(* CoDeSys 2.3.9.41 project: Mixer1_CFC_IL_LD_SFC_ST_v8.pro *)
(* Libraries: Standard.lib 4.10.05 12:14:46, IecSfc.lib 13.4.06 16:51:28, SYSLIBCALLBACK.LIB 26.9.08 17:43:52 *)

(* Task configuration *)
TASK NewTask (PRIORITY := 1); (* freewheeling *)
	VIS_PRG();
	PLC_Timers();
	PLC_ST_PRG();
END_TASK

(* Global variable list: Global_Variables *)
VAR_GLOBAL  (* 13 входов на 14 выходов + всп. пер. + входы и выходы таймеров  *)
(* Входы *)
    (* Кнопки Push Buttons -- префикс pb *)
	pbStrt: BOOL;             (* кнопка "Пуск"                                  *)
    pbStop: BOOL;             (* кнопка "Стоп"                                  *)
	pbCmpl: BOOL;             (* кнопка "Завершение работы"                     *)
	(* Кнопки-переключатели Switch Buttons -- префикс sb *)
	sbEVlv: BOOL;             (* переключатель "Открыть аварийный клапан"       *)
    (* Датчики Sensors -- префикс s *)
	sT1, _sT1: BOOL;          (* датчик нулевого уровня бака 1                  *)
	sT2, _sT2: BOOL;          (* датчик нулевого уровня бака 2                  *)
	sL0      : BOOL;          (* датчик уровня 0 резервуара                     *)
	sL1      : BOOL;          (* датчик уровня 1 резервуара                     *)
	sL2      : BOOL;          (* датчик уровня 2 резервуара                     *)
	sM,  _sM : BOOL;          (* датчик работы привода мешалки                  *)
	sUT      : BOOL;          (* датчик верхней температуры нагревателя         *)
	sLT      : BOOL;          (* датчик нижней  температуры нагревателя         *)
	sWT, _sWT: BOOL;          (* датчик рабочей температуры нагревателя         *)
(* Выходы *)
	(* Клапаны/Лампы Valves/Lamps -- префикс vlv/lmp *)
	vlv1, _vlv1: BOOL;        (* открыть клапан 1                               *)
	vlv2, _vlv2: BOOL;        (* открыть клапан 2                               *)
	vlvP       : BOOL;        (* открыть разливной клапан                       *)
	vlvE, _vlvE: BOOL;        (* открыть аварийный клапан                       *)
	(* Приводы/Лампы Actuators/Lamps -- префикс act/lmp *)
 	actHtr, _actHtr: BOOL;    (* включить нагреватель                           *)
	actMtr, _actMtr: BOOL;    (* запустить привод мешалки                       *)
    (* Режимы/Состояния/Лампы Modes/States/Lamps -- префикс m/q/lmp *)
	mSysOn,  _mSysOn : BOOL;  (* система включена                               *)
	mCompl,  _mCompl : BOOL;  (* режим плавного завершения работы установки     *)
    mMxIsFn, _mMxIsFn: BOOL;  (* смесь приготовлена                             *)
    mMxIsBd, _mMxIsBd: BOOL;  (* смесь испорчена                                *)
    mC1InMx, _mC1InMx: BOOL;  (* в смеси есть компонент 1                       *)
    mC2InMx, _mC2InMx: BOOL;  (* в смеси есть компонент 2                       *)
    (* Ошибки/Лампы Errors/Lamps -- префикс err/lmp *)
	errHtr, _errHtr: BOOL;    (* сигнал ошибки нагревателя                      *)
	errMtr, _errMtr: BOOL;    (* сигнал ошибки привода мешалки                  *)
(* Вспомогательные переменные Conditions -- префикс c *)
	cFin: BOOL;               (* условие завершения работы установки            *)
(* Таймеры Timers -- префикс tmr *)
	tmrMtr: TON := (PT := T#2s);    (* таймер ожидания запуска мешалки          *)
    tmrMix: TON := (PT := T#7s);    (* таймер работы мешалки                    *)
    tmrHtr: TON := (PT := T#12s);   (* таймер ожидания нагрева                  *)
END_VAR

(* POU VIS_PRG, ST *)
PROGRAM VIS_PRG
VAR
  (* ------- Обычные кнопки ------- *)
  PBTnk1: BOOL;                  (* наполнить бак 1 (синий)                *)
  PBTnk2: BOOL;                  (* наполнить бак 2 (красный)              *)
  PBCmp1: BOOL;                  (* осушить бак 1                          *)
  PBCmp2: BOOL;                  (* осушить бак 2                          *)
  (* ------- Кнопки-переключатели ------- *)
  SBMtrBrk: BOOL;                (* поломка привода мешалки                *)
  SBHtrBrk: BOOL;                (* поломка нагревателя                    *)
  (* ------- Жидкости ------- *)
  Cmp1, _Cmp1: INT;              (* объем компонента 1 (синего)   в баке 1 *)
  Cmp2, _Cmp2: INT;              (* объем компонента 2 (красного) в баке 2 *)
  Mix,   _Mix: INT;              (* объем смеси в резервуаре               *)
  MixClr:      DWORD;            (* цвет  смеси в резервуаре               *)
  Red,   _Red: REAL;             (* коэффициент красного цвета в смеси     *)
  (* ------- Нагреватель ------- *)
  HtrClr: DWORD:=16#00_FF_FF_FF; (* температура нагревателя (цвет)         *)
  HtrRed, _HtrRed: BYTE;         (* степень накаливания нагревателя        *)
  HtrOn: BOOL;                   (* нагреватель функционирует (греет)      *)
END_VAR
(* объем каждого из баков --- 300 единиц *)
(* пропускная способность каждого клапана равняется 1 единице за время прохода рабочего цикла ПЛК *)
(* но отрисовывать уменьшение объема жидкости в баке нужно в 3 раза медленне, чем происходит отрисовка заполнеия резервуара для смешивания *)
(* считается, что все клапаны обладают одинаковой пропускной способностью *)
Cmp1:= MAX(0,MIN(360,BOOL_TO_INT(NOT PBCmp1)*_Cmp1+BOOL_TO_INT(PBTnk1)*360-BOOL_TO_INT(vlv1)));
Cmp2:= MAX(0,MIN(240,BOOL_TO_INT(NOT PBCmp2)*_Cmp2+BOOL_TO_INT(PBTnk2)*240-BOOL_TO_INT(vlv2)));
Mix := MAX(0,_Mix
             +BOOL_TO_INT(vlv1 AND _Cmp1>0)
             +BOOL_TO_INT(vlv2 AND _Cmp2>0)
             -BOOL_TO_INT(vlvE AND _Mix >0)
             -BOOL_TO_INT(vlvP AND _Mix >0)
          );
Red := BOOL_TO_INT(Mix>0)*(_Red*_Mix+1*BOOL_TO_INT(vlv2 AND _Cmp2>0)
                                    -1*_Red*BOOL_TO_INT(vlvP AND _Mix >0)
                                    -1*_Red*BOOL_TO_INT(vlvE AND _Mix >0)
                                                                         )/MAX(1,Mix);
MixClr := 65536*REAL_TO_BYTE(255*(1-Red))+REAL_TO_BYTE(255*Red);
(* ------- Нагреватель ------- *)
HtrOn:=actHtr AND NOT SBHtrBrk; (* нагреватель включается, если не сломан       *)
HtrRed:=_HtrRed+BOOL_TO_BYTE(HtrOn AND _HtrRed<255)-BOOL_TO_BYTE(NOT HtrOn AND _HtrRed>0);
HtrClr:=65536*(255-HtrRed)+256*(255-HtrRed)+255;
(* ------- Выставление сигналов датчиков ------- *)
sT1:=(Cmp1>0);                  (* датчик нулевого уровня бака 1                *)
sT2:=(Cmp2>0);                  (* датчик нулевого уровня бака 2                *)
sL0:=(Mix>0);                   (* датчик уровня 0 резервуара                   *)
sL1:=(Mix>=180);                (* датчик уровня 1 резервуара                   *)
sL2:=(Mix>=300);                (* датчик уровня 2 резервуара                   *)
sM := NOT SBMtrBrk AND actMtr;  (* привод мешалки включается, если не сломан    *)
sUT:=(HtrRed>=252);
sLT:=(HtrRed>=160);
sWT:=(HtrRed>=150);
(* -------  Псевдооператорный раздел ------- *)
_Cmp1:=Cmp1; _Cmp2:=Cmp2; _Mix:=Mix; _Red:=Red; _HtrRed:=HtrRed;
END_PROGRAM

(* POU PLC_Timers, FBD *)
PROGRAM PLC_Timers
VAR
END_VAR
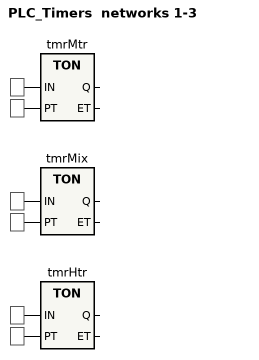
_FBD_ (* Function Block Diagram *)
NETWORK 1
	tmrMtr:TON(IN: , PT: )
NETWORK 2
	tmrMix:TON(IN: , PT: )
NETWORK 3
	tmrHtr:TON(IN: , PT: )
_END_FBD_
END_PROGRAM

(* POU PLC_ST_PRG, ST *)
PROGRAM PLC_ST_PRG
VAR
END_VAR
(* ------- Ошибки/Лампы ------- *)
IF NOT _errHtr AND NOT sWT AND (tmrHtr.Q OR _actHtr AND _sWT) THEN errHtr:=1;         (* errHtr+  *)
ELSIF  _errHtr AND pbStop                                     THEN errHtr:=0;         (* errHtr-  *)
END_IF;
IF NOT _errMtr AND NOT sM AND (tmrMtr.Q OR _actMtr AND _sM) THEN errMtr:=1;           (* errMtr+  *)
ELSIF  _errMtr AND pbStop                                   THEN errMtr:=0;           (* errMtr-  *)
END_IF;
(* ------- Режимы/Состояния/Лампы ------- *)
IF NOT _mMxIsBd AND     sL0 AND _vlvE AND _mC2InMx AND NOT _mMxIsFn THEN mMxIsBd:=1;  (* mMxIsBd+ *)
ELSIF  _mMxIsBd AND NOT sL0                                         THEN mMxIsBd:=0;  (* mMxIsBd- *)
END_IF;
IF NOT _mMxIsFn AND     sL0 AND NOT mMxIsBd AND tmrMix.Q THEN mMxIsFn:=1;             (* mMxIsFn+ *)
ELSIF  _mMxIsFn AND NOT sL0                              THEN mMxIsFn:=0;             (* mMxIsFn- *)
END_IF;
IF NOT _mC1InMx AND     sL0 AND _vlv1 AND _sT1 THEN mC1InMx:=1;                       (* mC1InMx+ *)
ELSIF  _mC1InMx AND NOT sL0                    THEN mC1InMx:=0;                       (* mC1InMx- *)
END_IF;
IF NOT _mC2InMx AND     sL0 AND _vlv2 AND _sT2 THEN mC2InMx:=1;                       (* mC2InMx+ *)
ELSIF  _mC2InMx AND NOT sL0                    THEN mC2InMx:=0;                       (* mC2InMx- *)
END_IF;
(* ------- Вспомогательные переменные ------- *)
cFin:= _mCompl AND NOT _vlv1 AND NOT sL0
                OR errHtr OR errMtr OR mMxIsBd OR sbEVlv OR pbStop
                OR NOT sT1 AND NOT sL1 AND NOT mMxIsFn
                OR NOT sT2 AND NOT sL2 AND NOT mMxIsFn;                               (* cFin     *)
(* ------- Режимы/Состояния/Лампы ------- *)
IF NOT _mSysOn AND pbStrt AND NOT cFin THEN mSysOn:=1;                                (* mSysOn+  *)
ELSIF  _mSysOn AND                cFin THEN mSysOn:=0;                                (* mSysOn-  *)
END_IF;
IF NOT _mCompl AND     mSysOn AND pbCmpl THEN mCompl:=1;                              (* mCompl+  *)
ELSIF  _mCompl AND NOT mSysOn            THEN mCompl:=0;                              (* mCompl-  *)
END_IF;
(* ------- Нагреватель/Лампа ------- *)
IF NOT _actHtr AND      mSysOn AND NOT sLT  THEN actHtr:=1;                           (* actHtr+  *)
ELSIF  _actHtr AND (NOT mSysOn OR      sUT) THEN actHtr:=0;                           (* actHtr-  *)
END_IF;
(* ------- Клапаны/Приводы/Лампы ------- *)
vlv1:=mSysOn AND sT1 AND NOT sL1               AND NOT mC2InMx AND sWT;               (* vlv1     *)
Vlv2:=mSysOn AND sT2 AND     sL1   AND NOT sL2 AND NOT mMxIsFn AND sWT;               (* vlv2     *)
actMtr:=mSysOn AND mC1InMx AND mC2InMx AND sL2 AND NOT mMxIsFn AND sWT;               (* actMtr   *)
vlvP:=mSysOn AND mMxIsFn;                                                             (* vlvP     *)
vlvE:=sbEVlv;                                                                         (* vlvE     *)
(* ------- Раздел таймеров ------- *)
tmrHtr.IN:= actHtr AND NOT sWT;                                                      (* tmrHtr.IN *)
tmrMtr.IN:= actMtr AND NOT sM;                                                       (* tmrMtr.IN *)
tmrMix.IN:= actMtr AND     sM;                                                       (* tmrMix.IN *)
(* ------- Псевдооператорный раздел ------- *)
_errMtr:=errMtr; _errHtr:=errHtr;
_mC1InMx:=mC1InMx; _mC2InMx:=mC2InMx;
_mMxIsFn:=mMxIsFn; _mMxIsBd:=mMxIsBd;
_mSysOn:=mSysOn; _mCompl:=mCompl;
_vlvE:=vlvE; _vlv1:=vlv1; _vlv2:=vlv2;
_actHtr:=actHtr; _actMtr:=actMtr;
_sT1:=sT1; _sT2:=sT2; _sM :=sM; _sWT:=sWT;
END_PROGRAM

(* POU PLC_CFC_PRG, FAI *)
PROGRAM PLC_CFC_PRG
VAR
END_VAR
(* body not read: cfc101 *)
END_PROGRAM

(* POU PLC_IL_PRG, IL *)
PROGRAM PLC_IL_PRG
VAR
END_VAR
	(* ------- Ошибки/Лампы ------- *)
	(* IF      *)
	LDN		_errHtr							(* errHtr  *)
	ANDN	sWT
	AND		(tmrHtr.Q
	OR		(_actHtr
	AND		_sWT
	)
	)
	S		errHtr		(* errHtr:=1 *)
	LD		_errHtr		(* ELSIF     *)
	AND		pbStop
	R		errHtr		(* errHtr:=0 *)
	(* END_IF  *)
	(* ------- *)
	(* IF      *)
	LDN		_errMtr							(* errMtr  *)
	ANDN	sM
	AND		(tmrMtr.Q
	OR		(_actMtr
	AND		_sM
	)
	)
	S		errMtr		(* errMtr:=1 *)
	LD		_errMtr		(* ELSIF     *)
	AND		pbStop
	R		errMtr		(* errMtr:=0 *)
	(* END_IF  *)
	(* ------- Режимы/Состояния/Лампы ------- *)
	(* IF      *)
	LDN		_mMxIsBd						(* mMxIsBd *)
	AND		sL0
	AND		_vlvE
	AND		_mC2InMx
	ANDN	_mMxIsFn
	S		mMxIsBd		(* mMxIsBd:=1 *)
	LD		_mMxIsBd	(* ELSIF      *)
	ANDN	sL0
	R		mMxIsBd 	(* mMxIsBd:=0 *)
	(* END_IF  *)
	(* ------- *)
	(* IF      *)
	LDN		_mMxIsFn						(* mMxIsFn *)
	AND		sL0
	ANDN	mMxIsBd
	AND		tmrMix.Q
	S		mMxIsFn		(* mMxIsFn:=1 *)
	LD		_mMxIsFn	(* ELSIF      *)
	ANDN	sL0
	R		mMxIsFn		(* mMxIsFn:=0 *)
	(* END_IF  *)
	(* ------- *)
	(* IF      *)
	LDN		_mC1InMx						(* mC1InMx *)
	AND		sL0
	AND		_vlv1
	AND		_sT1
	S		mC1InMx		(* mC1InMx:=1 *)
	LD		_mC1InMx	(* ELSIF      *)
	ANDN	sL0
	R		mC1InMx		(* mC1InMx:=0 *)
	(* END_IF  *)
	(* ------- *)
	(* IF      *)
	LDN		_mC2InMx						(* mC2InMx *)
	AND		sL0
	AND		_vlv2
	AND		_sT2
	S		mC2InMx		(* mC2InMx:=1 *)
	LD		_mC2InMx	(* ELSIF      *)
	ANDN	sL0
	R		mC2InMx		(* mC2InMx:=0 *)
	(* END_IF  *)
	(* ------- Вспомогательные переменные ------- *)
	LD		_mCompl							(* cFin    *)
	ANDN	_vlv1
	ANDN	sL0
	OR		errHtr
	OR		errMtr
	OR		mMxIsBd
	OR		sbEVlv
	OR		pbStop
	OR		(sT1
	NOT
	ANDN	sL1
	ANDN	mMxIsFn
	)
	OR		(sT2
	NOT
	ANDN	sL2
	ANDN	mMxIsFn
	)
	ST		cFin
	(* ------- Режимы/Состояния/Лампы ------- *)
	(* IF      *)
	LDN		_mSysOn							(* mSysOn  *)
	AND		pbStrt
	ANDN	cFin
	S		mSysOn		(* mSysOn:=1 *)
	LD		_mSysOn		(* ELSIF     *)
	AND		cFin
	R		mSysOn		(* mSysOn:=0 *)
	(* END_IF  *)
	(* ------- *)
	(* IF      *)
	LDN		_mCompl							(* mCompl  *)
	AND		mSysOn
	AND		pbCmpl
	S		mCompl		(* mCompl:=1 *)
	LD		_mCompl		(* ELSIF     *)
	ANDN	mSysOn
	R		mCompl		(* mCompl:=0 *)
	(* END_IF  *)
	(* ------- Нагреватель/Лампа ------- *)
	(* IF      *)
	LDN		_actHtr							(* actHtr  *)
	AND		mSysOn
	ANDN	sLT
	S		actHtr		(* actHtr:=1 *)
	LD		_actHtr		(* ELSIF     *)
	AND		(mSysOn
	NOT
	OR		sUT
	)
	R		actHtr		(* actHtr:=0 *)
	(* END_IF  *)
	(* ------- Клапаны/Лампы ------- *)
	LD		mSysOn 						    (* Vlv1    *)
	AND		sT1
	ANDN	sL1
	ANDN	mC2InMx
	AND		sWT
	ST		vlv1
	(* ------- Клапаны/Лампы ------- *)
	LD		mSysOn 							(* Vlv2    *)
	AND		sT2
	AND		sL1
	ANDN	sL2
	ANDN	mMxIsFn
	AND		sWT
	ST		vlv2
	(* ------- Приводы/Лампы ------- *)
	LD		mSysOn							(* actMtr  *)
	AND		mC1InMx
	AND		mC2InMx
	AND		sL2
	ANDN	mMxIsFn
	AND		sWT
	ST		actMtr
	(* ------- Клапаны/Лампы ------- *)
	LD		mSysOn							(* vlvP    *)
	AND		mMxIsFn
	ST		vlvP
	(* ------- *)
	LD		sbEVlv							(* vlvE    *)
	ST		vlvE
	(* ------- Раздел таймеров ------- *)
	LD		actHtr						  (* tmrHtr.IN *)
	ANDN	sWT
	ST		tmrHtr.IN
	(* ------- *)
	LD		actMtr						  (* tmrMtr.IN *)
	ANDN	sM
	ST		tmrMtr.IN
	(* ------- *)
	LD		actMtr						  (* tmrMix.IN *)
	AND		sM
	ST		tmrMix.IN
	(* ------- Псевдооператорный раздел ------- *)
	(* ------- Ошибки ------- *)
	LD		errMtr
	ST		_errMtr		(* _errMtr:=errMtr;   *)
	LD		errHtr
	ST		_errHtr		(* _errHtr:=errHtr;   *)
	(* ------- Режимы/Состояния ------- *)
	LD		mC1InMx
	ST		_mC1InMx	(* _mC1InMx:=mC1InMx; *)
	LD		mC2InMx
	ST		_mC2InMx	(* _mC2InMx:=mC2InMx; *)
	LD		mMxIsFn
	ST		_mMxIsFn	(* _mMxIsFn:=mMxIsFn; *)
	LD		mMxIsBd
	ST		_mMxIsBd	(* _mMxIsBd:=mMxIsBd; *)
	LD		mSysOn
	ST		_mSysOn		(* _mSysOn:=mSysOn;   *)
	LD		mCompl
	ST		_mCompl		(* _mCompl:=mCompl;   *)
	(* ------- Клапаны ------- *)
	LD		vlvE
	ST		_vlvE		(* _vlvE:=vlvE;       *)
	LD		vlv1
	ST		_vlv1		(* _vlv1:=vlv1;       *)
	LD		vlv2
	ST		_vlv2		(* _vlv2:=vlv2;       *)
	(* ------- Приводы ------- *)
	LD		actHtr
	ST		_actHtr		(* _actHtr:=actHtr;   *)
	LD		actMtr
	ST		_actMtr		(* _actMtr:=actMtr;   *)
	(* ------- Датчики ------- *)
	LD		sT1
	ST		_sT1		(* _sT1:=sT1;         *)
	LD		sT2
	ST		_sT2		(* _sT2:=sT2;         *)
	LD		sM
	ST		_sM			(* _sM:=sM;           *)
	LD		sWT
	ST		_sWT		(* _sWT:=sWT;         *)
END_PROGRAM

(* POU PLC_LD_PRG, LD *)
PROGRAM PLC_LD_PRG
VAR
END_VAR
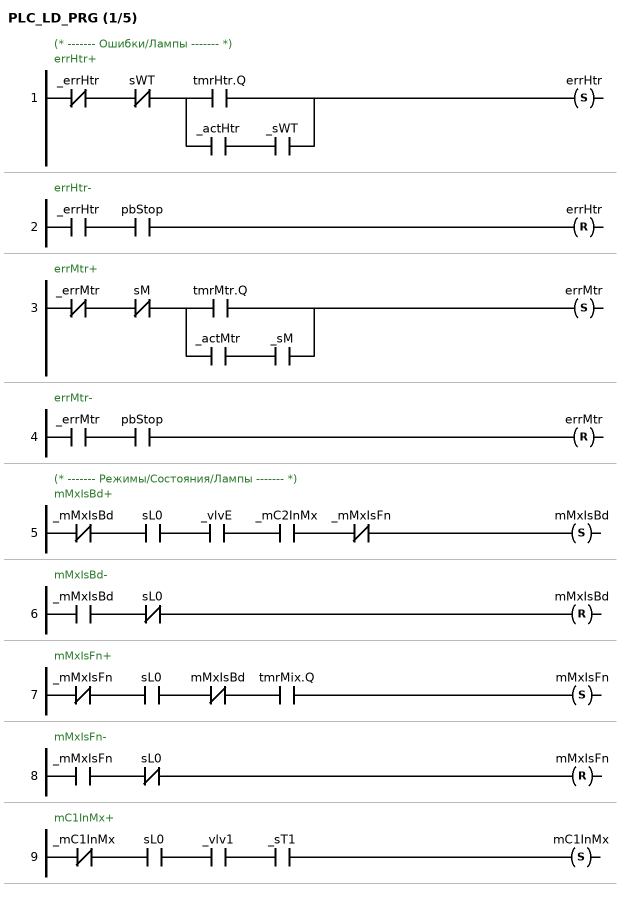
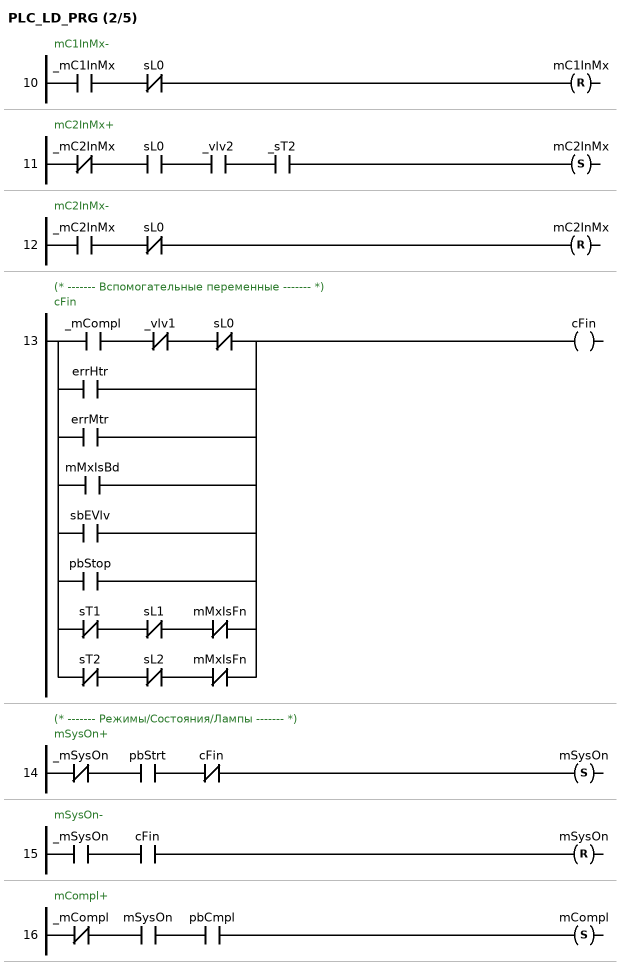
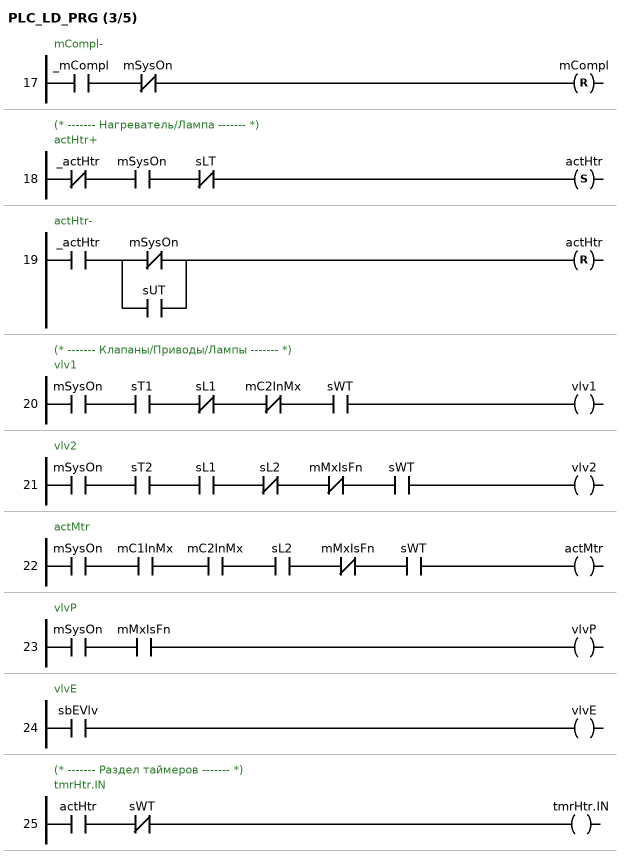
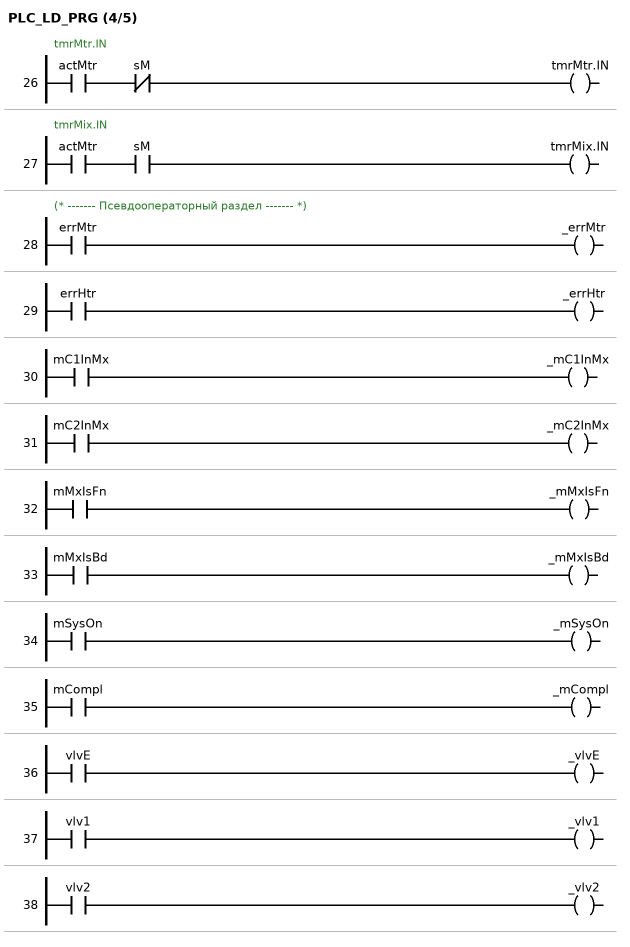
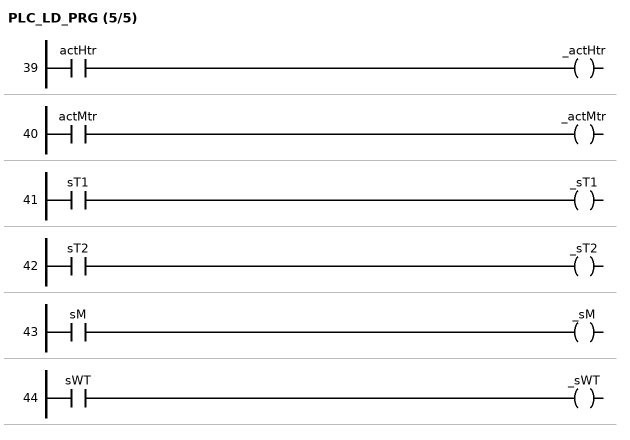
_LD_ (* Ladder Diagram *)
NETWORK 1 (* ( * ------- Ошибки/Лампы ------- * ) / errHtr+ *)
	[/_errHtr] - [/sWT] - { [tmrHtr.Q] | [_actHtr] - [_sWT] } --- (S errHtr)
NETWORK 2 (* errHtr- *)
	[_errHtr] - [pbStop] --- (R errHtr)
NETWORK 3 (* errMtr+ *)
	[/_errMtr] - [/sM] - { [tmrMtr.Q] | [_actMtr] - [_sM] } --- (S errMtr)
NETWORK 4 (* errMtr- *)
	[_errMtr] - [pbStop] --- (R errMtr)
NETWORK 5 (* ( * ------- Режимы/Состояния/Лампы ------- * ) / mMxIsBd+ *)
	[/_mMxIsBd] - [sL0] - [_vlvE] - [_mC2InMx] - [/_mMxIsFn] --- (S mMxIsBd)
NETWORK 6 (* mMxIsBd- *)
	[_mMxIsBd] - [/sL0] --- (R mMxIsBd)
NETWORK 7 (* mMxIsFn+ *)
	[/_mMxIsFn] - [sL0] - [/mMxIsBd] - [tmrMix.Q] --- (S mMxIsFn)
NETWORK 8 (* mMxIsFn- *)
	[_mMxIsFn] - [/sL0] --- (R mMxIsFn)
NETWORK 9 (* mC1InMx+ *)
	[/_mC1InMx] - [sL0] - [_vlv1] - [_sT1] --- (S mC1InMx)
NETWORK 10 (* mC1InMx- *)
	[_mC1InMx] - [/sL0] --- (R mC1InMx)
NETWORK 11 (* mC2InMx+ *)
	[/_mC2InMx] - [sL0] - [_vlv2] - [_sT2] --- (S mC2InMx)
NETWORK 12 (* mC2InMx- *)
	[_mC2InMx] - [/sL0] --- (R mC2InMx)
NETWORK 13 (* ( * ------- Вспомогательные переменные ------- * ) / cFin *)
	{ [_mCompl] - [/_vlv1] - [/sL0] | [errHtr] | [errMtr] | [mMxIsBd] | [sbEVlv] | [pbStop] | [/sT1] - [/sL1] - [/mMxIsFn] | [/sT2] - [/sL2] - [/mMxIsFn] } --- (cFin)
NETWORK 14 (* ( * ------- Режимы/Состояния/Лампы ------- * ) / mSysOn+ *)
	[/_mSysOn] - [pbStrt] - [/cFin] --- (S mSysOn)
NETWORK 15 (* mSysOn- *)
	[_mSysOn] - [cFin] --- (R mSysOn)
NETWORK 16 (* mCompl+ *)
	[/_mCompl] - [mSysOn] - [pbCmpl] --- (S mCompl)
NETWORK 17 (* mCompl- *)
	[_mCompl] - [/mSysOn] --- (R mCompl)
NETWORK 18 (* ( * ------- Нагреватель/Лампа ------- * ) / actHtr+ *)
	[/_actHtr] - [mSysOn] - [/sLT] --- (S actHtr)
NETWORK 19 (* actHtr- *)
	[_actHtr] - { [/mSysOn] | [sUT] } --- (R actHtr)
NETWORK 20 (* ( * ------- Клапаны/Приводы/Лампы ------- * ) / vlv1 *)
	[mSysOn] - [sT1] - [/sL1] - [/mC2InMx] - [sWT] --- (vlv1)
NETWORK 21 (* vlv2 *)
	[mSysOn] - [sT2] - [sL1] - [/sL2] - [/mMxIsFn] - [sWT] --- (vlv2)
NETWORK 22 (* actMtr *)
	[mSysOn] - [mC1InMx] - [mC2InMx] - [sL2] - [/mMxIsFn] - [sWT] --- (actMtr)
NETWORK 23 (* vlvP *)
	[mSysOn] - [mMxIsFn] --- (vlvP)
NETWORK 24 (* vlvE *)
	[sbEVlv] --- (vlvE)
NETWORK 25 (* ( * ------- Раздел таймеров ------- * ) / tmrHtr.IN *)
	[actHtr] - [/sWT] --- (tmrHtr.IN)
NETWORK 26 (* tmrMtr.IN *)
	[actMtr] - [/sM] --- (tmrMtr.IN)
NETWORK 27 (* tmrMix.IN *)
	[actMtr] - [sM] --- (tmrMix.IN)
NETWORK 28 (* ( * ------- Псевдооператорный раздел ------- * ) *)
	[errMtr] --- (_errMtr)
NETWORK 29
	[errHtr] --- (_errHtr)
NETWORK 30
	[mC1InMx] --- (_mC1InMx)
NETWORK 31
	[mC2InMx] --- (_mC2InMx)
NETWORK 32
	[mMxIsFn] --- (_mMxIsFn)
NETWORK 33
	[mMxIsBd] --- (_mMxIsBd)
NETWORK 34
	[mSysOn] --- (_mSysOn)
NETWORK 35
	[mCompl] --- (_mCompl)
NETWORK 36
	[vlvE] --- (_vlvE)
NETWORK 37
	[vlv1] --- (_vlv1)
NETWORK 38
	[vlv2] --- (_vlv2)
NETWORK 39
	[actHtr] --- (_actHtr)
NETWORK 40
	[actMtr] --- (_actMtr)
NETWORK 41
	[sT1] --- (_sT1)
NETWORK 42
	[sT2] --- (_sT2)
NETWORK 43
	[sM] --- (_sM)
NETWORK 44
	[sWT] --- (_sWT)
_END_LD_
(* the same logic as Structured Text *)
(* Network 1: ( * ------- Ошибки/Лампы ------- * ) / errHtr+ *)
IF NOT _errHtr AND NOT sWT AND (tmrHtr.Q OR _actHtr AND _sWT) THEN errHtr := TRUE; END_IF;
(* Network 2: errHtr- *)
IF _errHtr AND pbStop THEN errHtr := FALSE; END_IF;
(* Network 3: errMtr+ *)
IF NOT _errMtr AND NOT sM AND (tmrMtr.Q OR _actMtr AND _sM) THEN errMtr := TRUE; END_IF;
(* Network 4: errMtr- *)
IF _errMtr AND pbStop THEN errMtr := FALSE; END_IF;
(* Network 5: ( * ------- Режимы/Состояния/Лампы ------- * ) / mMxIsBd+ *)
IF NOT _mMxIsBd AND sL0 AND _vlvE AND _mC2InMx AND NOT _mMxIsFn THEN mMxIsBd := TRUE; END_IF;
(* Network 6: mMxIsBd- *)
IF _mMxIsBd AND NOT sL0 THEN mMxIsBd := FALSE; END_IF;
(* Network 7: mMxIsFn+ *)
IF NOT _mMxIsFn AND sL0 AND NOT mMxIsBd AND tmrMix.Q THEN mMxIsFn := TRUE; END_IF;
(* Network 8: mMxIsFn- *)
IF _mMxIsFn AND NOT sL0 THEN mMxIsFn := FALSE; END_IF;
(* Network 9: mC1InMx+ *)
IF NOT _mC1InMx AND sL0 AND _vlv1 AND _sT1 THEN mC1InMx := TRUE; END_IF;
(* Network 10: mC1InMx- *)
IF _mC1InMx AND NOT sL0 THEN mC1InMx := FALSE; END_IF;
(* Network 11: mC2InMx+ *)
IF NOT _mC2InMx AND sL0 AND _vlv2 AND _sT2 THEN mC2InMx := TRUE; END_IF;
(* Network 12: mC2InMx- *)
IF _mC2InMx AND NOT sL0 THEN mC2InMx := FALSE; END_IF;
(* Network 13: ( * ------- Вспомогательные переменные ------- * ) / cFin *)
cFin := _mCompl AND NOT _vlv1 AND NOT sL0 OR errHtr OR errMtr OR mMxIsBd OR sbEVlv OR pbStop OR NOT sT1 AND NOT sL1 AND NOT mMxIsFn OR NOT sT2 AND NOT sL2 AND NOT mMxIsFn;
(* Network 14: ( * ------- Режимы/Состояния/Лампы ------- * ) / mSysOn+ *)
IF NOT _mSysOn AND pbStrt AND NOT cFin THEN mSysOn := TRUE; END_IF;
(* Network 15: mSysOn- *)
IF _mSysOn AND cFin THEN mSysOn := FALSE; END_IF;
(* Network 16: mCompl+ *)
IF NOT _mCompl AND mSysOn AND pbCmpl THEN mCompl := TRUE; END_IF;
(* Network 17: mCompl- *)
IF _mCompl AND NOT mSysOn THEN mCompl := FALSE; END_IF;
(* Network 18: ( * ------- Нагреватель/Лампа ------- * ) / actHtr+ *)
IF NOT _actHtr AND mSysOn AND NOT sLT THEN actHtr := TRUE; END_IF;
(* Network 19: actHtr- *)
IF _actHtr AND (NOT mSysOn OR sUT) THEN actHtr := FALSE; END_IF;
(* Network 20: ( * ------- Клапаны/Приводы/Лампы ------- * ) / vlv1 *)
vlv1 := mSysOn AND sT1 AND NOT sL1 AND NOT mC2InMx AND sWT;
(* Network 21: vlv2 *)
vlv2 := mSysOn AND sT2 AND sL1 AND NOT sL2 AND NOT mMxIsFn AND sWT;
(* Network 22: actMtr *)
actMtr := mSysOn AND mC1InMx AND mC2InMx AND sL2 AND NOT mMxIsFn AND sWT;
(* Network 23: vlvP *)
vlvP := mSysOn AND mMxIsFn;
(* Network 24: vlvE *)
vlvE := sbEVlv;
(* Network 25: ( * ------- Раздел таймеров ------- * ) / tmrHtr.IN *)
tmrHtr.IN := actHtr AND NOT sWT;
(* Network 26: tmrMtr.IN *)
tmrMtr.IN := actMtr AND NOT sM;
(* Network 27: tmrMix.IN *)
tmrMix.IN := actMtr AND sM;
(* Network 28: ( * ------- Псевдооператорный раздел ------- * ) *)
_errMtr := errMtr;
(* Network 29 *)
_errHtr := errHtr;
(* Network 30 *)
_mC1InMx := mC1InMx;
(* Network 31 *)
_mC2InMx := mC2InMx;
(* Network 32 *)
_mMxIsFn := mMxIsFn;
(* Network 33 *)
_mMxIsBd := mMxIsBd;
(* Network 34 *)
_mSysOn := mSysOn;
(* Network 35 *)
_mCompl := mCompl;
(* Network 36 *)
_vlvE := vlvE;
(* Network 37 *)
_vlv1 := vlv1;
(* Network 38 *)
_vlv2 := vlv2;
(* Network 39 *)
_actHtr := actHtr;
(* Network 40 *)
_actMtr := actMtr;
(* Network 41 *)
_sT1 := sT1;
(* Network 42 *)
_sT2 := sT2;
(* Network 43 *)
_sM := sM;
(* Network 44 *)
_sWT := sWT;
END_PROGRAM

(* POU PLC_SFC_PRG, SFC *)
PROGRAM PLC_SFC_PRG
VAR
END_VAR
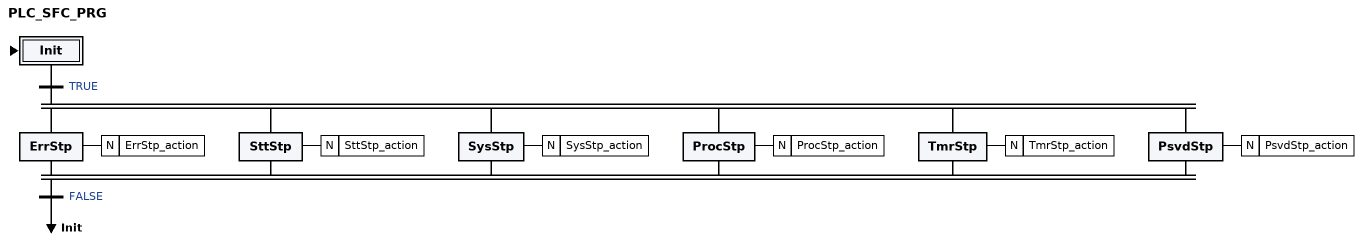
INITIAL_STEP Init:
END_STEP
TRANSITION FROM Init TO (ErrStp, SttStp, SysStp, ProcStp, TmrStp, PsvdStp) := TRUE;
END_TRANSITION
STEP ErrStp:
	ErrStp_action(N);
END_STEP
STEP SttStp:
	SttStp_action(N);
END_STEP
STEP SysStp:
	SysStp_action(N);
END_STEP
STEP ProcStp:
	ProcStp_action(N);
END_STEP
STEP TmrStp:
	TmrStp_action(N);
END_STEP
STEP PsvdStp:
	PsvdStp_action(N);
END_STEP
TRANSITION FROM (ErrStp, SttStp, SysStp, ProcStp, TmrStp, PsvdStp) TO Init := FALSE;
END_TRANSITION

ACTION ErrStp_action:
(* ------- Состояния/Ошибки/Лампы ------- *)
IF NOT _errHtr AND NOT sWT AND (tmrHtr.Q OR _actHtr AND _sWT) THEN errHtr:=1;    (* errHtr+ *)
ELSIF  _errHtr AND pbStop                                     THEN errHtr:=0;    (* errHtr- *)
END_IF;
IF NOT _errMtr AND NOT sM AND (tmrMtr.Q OR _actMtr AND _sM) THEN errMtr:=1;      (* errMtr+ *)
ELSIF  _errMtr AND pbStop                                   THEN errMtr:=0;      (* MtrErr- *)
END_IF;
END_ACTION

ACTION SttStp_action:
(* ------- Состояния/Лампы ------- *)
IF NOT _mMxIsBd AND     sL0 AND _vlvE AND _mC2InMx AND NOT _mMxIsFn THEN mMxIsBd:=1; (* mMxIsBd+ *)
ELSIF  _mMxIsBd AND NOT sL0                                         THEN mMxIsBd:=0; (* mMxIsBd- *)
END_IF;
IF NOT _mMxIsFn AND     sL0 AND NOT mMxIsBd AND tmrMix.Q THEN mMxIsFn:=1;            (* mMxIsFn+ *)
ELSIF  _mMxIsFn AND NOT sL0                              THEN mMxIsFn:=0;            (* mMxIsFn- *)
END_IF;
IF NOT _mC1InMx AND     sL0 AND _vlv1 AND _sT1 THEN mC1InMx:=1;                      (* mC1InMx+ *)
ELSIF  _mC1InMx AND NOT sL0                    THEN mC1InMx:=0;                      (* mC1InMx- *)
END_IF;
IF NOT _mC2InMx AND     sL0 AND _vlv2 AND _sT2 THEN mC2InMx:=1;                      (* mC2InMx+ *)
ELSIF  _mC2InMx AND NOT sL0                    THEN mC2InMx:=0;                      (* mC2InMx- *)
END_IF;
END_ACTION

ACTION SysStp_action:
(* ------- Вспомогательные переменные ------- *)
cFin:= _mCompl AND NOT _vlv1 AND NOT sL0
                OR errHtr OR errMtr OR mMxIsBd OR sbEVlv OR pbStop
                OR NOT sT1 AND NOT sL1 AND NOT mMxIsFn
                OR NOT sT2 AND NOT sL2 AND NOT mMxIsFn;             (* cFin     *)
(* ------- Состояния/Лампы ------- *)
IF NOT _mSysOn AND pbStrt AND NOT cFin THEN mSysOn:=1;              (* mSysOn+  *)
ELSIF  _mSysOn AND                cFin THEN mSysOn:=0;              (* mSysOn-  *)
END_IF;
IF NOT _mCompl AND     mSysOn AND pbCmpl THEN mCompl:=1;            (* mCompl+  *)
ELSIF  _mCompl AND NOT mSysOn            THEN mCompl:=0;            (* mCompl-  *)
END_IF;
END_ACTION

ACTION ProcStp_action:
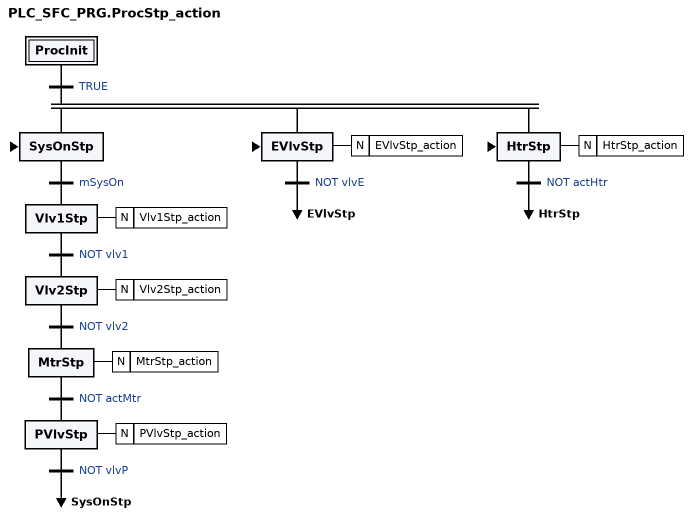
INITIAL_STEP ProcInit:
END_STEP
TRANSITION FROM ProcInit TO (SysOnStp, EVlvStp, HtrStp) := TRUE;
END_TRANSITION
STEP SysOnStp:
END_STEP
TRANSITION FROM SysOnStp TO Vlv1Stp := mSysOn;
END_TRANSITION
STEP Vlv1Stp:
	Vlv1Stp_action(N);
END_STEP
TRANSITION FROM Vlv1Stp TO Vlv2Stp := NOT vlv1;
END_TRANSITION
STEP Vlv2Stp:
	Vlv2Stp_action(N);
END_STEP
TRANSITION FROM Vlv2Stp TO MtrStp := NOT vlv2;
END_TRANSITION
STEP MtrStp:
	MtrStp_action(N);
END_STEP
TRANSITION FROM MtrStp TO PVlvStp := NOT actMtr;
END_TRANSITION
STEP EVlvStp:
	EVlvStp_action(N);
END_STEP
TRANSITION FROM EVlvStp TO EVlvStp := NOT vlvE;
END_TRANSITION
STEP HtrStp:
	HtrStp_action(N);
END_STEP
TRANSITION FROM HtrStp TO HtrStp := NOT actHtr;
END_TRANSITION
STEP PVlvStp:
	PVlvStp_action(N);
END_STEP
TRANSITION FROM PVlvStp TO SysOnStp := NOT vlvP;
END_TRANSITION

ACTION Vlv1Stp_action:
vlv1:=mSysOn AND sT1 AND NOT sL1 AND NOT mC2InMx AND sWT;            (* vlv1    *)
END_ACTION

ACTION Vlv2Stp_action:
vlv2:=mSysOn AND sT2 AND sL1 AND NOT sL2 AND NOT mMxIsFn AND sWT;            (* vlv2    *)
END_ACTION

ACTION MtrStp_action:
actMtr :=mSysOn AND mC1InMx AND mC2InMx AND sL2 AND NOT mMxIsFn AND sWT;            (* actMtr     *)
END_ACTION

ACTION EVlvStp_action:
vlvE:=sbEVlv;
END_ACTION

ACTION HtrStp_action:
(* ------- Нагреватель/Лампа ------- *)
IF NOT _actHtr AND      mSysOn AND NOT sLT  THEN actHtr:=1;            (* actHtr+    *)
ELSIF  _actHtr AND (NOT mSysOn OR      sUT) THEN actHtr:=0;            (* actHtr-    *)
END_IF;
END_ACTION

ACTION PVlvStp_action:
vlvP:=mSysOn AND mMxIsFn;            (* vlvP    *)
END_ACTION
END_ACTION

ACTION TmrStp_action:
(* ------- Раздел таймеров ------- *)
tmrHtr.IN:= actHtr AND NOT sWT;            (* tmrHtr.IN *)
tmrMtr.IN:= actMtr AND NOT sM;             (* tmrMtr.IN *)
tmrMix.IN:= actMtr AND     sM;             (* tmrMix.IN *)
END_ACTION

ACTION PsvdStp_action:
(* ------- Псевдооператорный раздел ------- *)
_errMtr:=errMtr; _errHtr:=errHtr;
_mC1InMx:=mC1InMx; _mC2InMx:=mC2InMx;
_mMxIsFn:=mMxIsFn; _mMxIsBd:=mMxIsBd;
_mSysOn:=mSysOn;   _mCompl:=mCompl;
_vlvE:=vlvE; _vlv1:=vlv1; _vlv2:=vlv2;
_actHtr:=actHtr; _actMtr:=actMtr;
_sT1:=sT1; _sT2:=sT2; _sM :=sM; _sWT:=sWT;
END_ACTION
END_PROGRAM

(* Visualisation Vis_Mixer
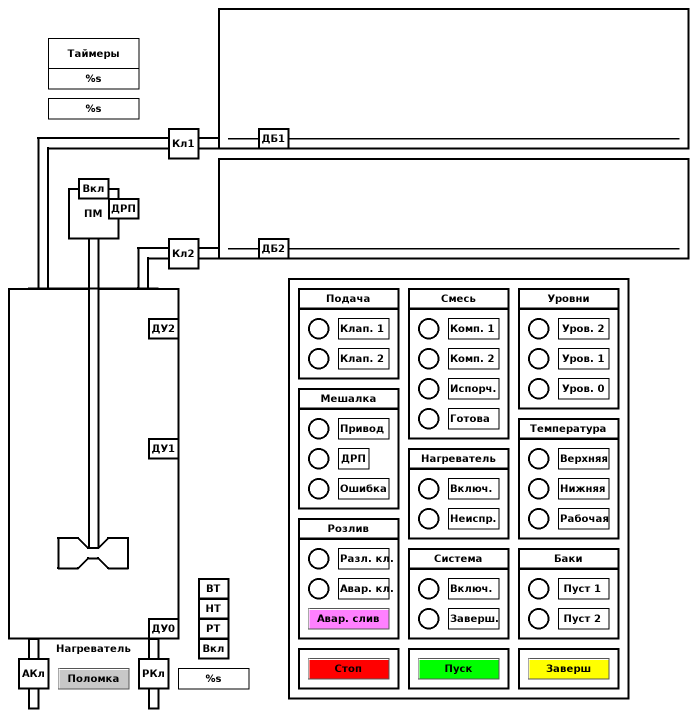
rounded rectangle at (250,20)-(721,161): taps VIS_PRG.PBTnk1
rectangle at (200,250)-(231,281): text "Кл2"; alarm colour if .vlv2
rectangle at (170,670)-(201,701): text "РКл"; alarm colour if .vlvP
rounded rectangle at (250,170)-(721,271): taps VIS_PRG.PBTnk2
rectangle at (200,140)-(231,171): text "Кл1"; alarm colour if .vlv1
rectangle at (260,260)-(711,261): taps VIS_PRG.PBCmp2; top -VIS_PRG.Cmp2/3
rectangle at (260,150)-(711,151): taps VIS_PRG.PBCmp1; top -VIS_PRG.Cmp1/3
rectangle at (50,670)-(81,701): text "АКл"; alarm colour if .vlvE
rectangle at (290,250)-(321,271): text "ДБ2"; alarm colour if .sT2
rectangle at (290,140)-(321,161): text "ДБ1"; alarm colour if .sT1
button at (340,620)-(421,641): text "Авар. слив"; toggles .sbEVlv
rectangle at (370,590)-(421,611): text "Авар. кл."
rectangle at (370,560)-(421,581): text "Разл. кл."
rectangle at (370,430)-(421,451): text "Привод"
rectangle at (370,490)-(421,511): text "Ошибка"
rectangle at (370,460)-(401,481): text "ДРП"
rectangle at (370,330)-(421,351): text "Клап. 1"
rectangle at (370,360)-(421,381): text "Клап. 2"
rectangle at (480,420)-(531,441): text "Готова"
rectangle at (480,390)-(531,411): text "Испорч."
ellipse at (340,590)-(361,611): alarm colour if .vlvE
ellipse at (340,560)-(361,581): alarm colour if .vlvP
ellipse at (340,430)-(361,451): alarm colour if .actMtr
ellipse at (340,460)-(361,481): alarm colour if .sM
ellipse at (340,490)-(361,511): alarm colour if .errMtr
ellipse at (340,360)-(361,381): alarm colour if .vlv2
ellipse at (340,330)-(361,351): alarm colour if .vlv1
ellipse at (450,390)-(471,411): alarm colour if .mMxIsBd
ellipse at (450,420)-(471,441): alarm colour if .mMxIsFn
rectangle at (120,210)-(131,561): alarm colour if .sM
polygon at (90,550)-(160,580): alarm colour if .sM
rectangle at (100,200)-(151,251): text "ПМ"; alarm colour if VIS_PRG.SBMtrBrk; toggles VIS_PRG.SBMtrBrk
rectangle at (140,210)-(171,231): text "ДРП"; alarm colour if .sM
rectangle at (110,190)-(141,211): text "Вкл"; alarm colour if .actMtr
rectangle at (480,330)-(531,351): text "Комп. 1"
rectangle at (480,360)-(531,381): text "Комп. 2"
ellipse at (450,330)-(471,351): alarm colour if .mC1InMx
ellipse at (450,360)-(471,381): alarm colour if .mC2InMx
rectangle at (590,590)-(641,611): text "Пуст 1"
rectangle at (590,620)-(641,641): text "Пуст 2"
ellipse at (560,590)-(581,611): alarm colour if NOT .sT1
ellipse at (560,620)-(581,641): alarm colour if NOT .sT2
rectangle at (590,390)-(641,411): text "Уров. 0"
rectangle at (590,360)-(641,381): text "Уров. 1"
rectangle at (590,330)-(641,351): text "Уров. 2"
ellipse at (560,390)-(581,411): alarm colour if .sL0
ellipse at (560,360)-(581,381): alarm colour if .sL1
ellipse at (560,330)-(581,351): alarm colour if .sL2
rectangle at (80,110)-(171,131): text "%s"; shows .tmrMtr.ET
rectangle at (80,50)-(171,81): text "Таймеры"
rectangle at (340,300)-(421,321): text "Подача"
rectangle at (450,300)-(531,321): text "Смесь"
rectangle at (340,400)-(421,421): text "Мешалка"
rectangle at (340,530)-(421,551): text "Розлив"
rectangle at (560,300)-(641,321): text "Уровни"
rectangle at (180,630)-(211,651): text "ДУ0"; alarm colour if .sL0
rectangle at (180,450)-(211,471): text "ДУ1"; alarm colour if .sL1
rectangle at (180,330)-(211,351): text "ДУ2"; alarm colour if .sL2
rectangle at (80,650)-(171,671): text "Нагреватель"
rectangle at (480,590)-(531,611): text "Включ."
rectangle at (480,620)-(531,641): text "Заверш."
ellipse at (450,590)-(471,611): alarm colour if .mSysOn
ellipse at (450,620)-(471,641): alarm colour if .mCompl
rectangle at (450,560)-(531,581): text "Система"
rectangle at (230,650)-(261,671): text "Вкл"; alarm colour if .actHtr
rectangle at (230,630)-(261,651): text "РТ"; alarm colour if .sWT
rectangle at (230,610)-(261,631): text "НТ"; alarm colour if .sLT
rectangle at (230,590)-(261,611): text "ВТ"; alarm colour if .sUT
button at (90,680)-(161,701): text "Поломка"; toggles VIS_PRG.SBHtrBrk
rectangle at (210,680)-(281,701): text "%s"; shows .tmrHtr.ET
rectangle at (80,80)-(171,101): text "%s"; shows .tmrMix.ET
rectangle at (480,490)-(531,511): text "Включ."
rectangle at (480,520)-(531,541): text "Неиспр."
ellipse at (450,490)-(471,511): alarm colour if .actHtr
ellipse at (450,520)-(471,541): alarm colour if .errHtr
rectangle at (450,460)-(531,481): text "Нагреватель"
rectangle at (590,460)-(641,481): text "Верхняя"
rectangle at (590,490)-(641,511): text "Нижняя"
ellipse at (560,460)-(581,481): alarm colour if .sUT
ellipse at (560,490)-(581,511): alarm colour if .sLT
rectangle at (560,430)-(641,451): text "Температура"
rectangle at (590,520)-(641,541): text "Рабочая"
ellipse at (560,520)-(581,541): alarm colour if .sWT
button at (450,670)-(531,691): text "Пуск"; taps .pbStrt
button at (560,670)-(641,691): text "Заверш"; taps .pbCmpl
button at (340,670)-(421,691): text "Стоп"; taps .pbStop
rectangle at (560,560)-(641,581): text "Баки"
28 more shapes without text or variables
2 elements of other kinds (tables, trends, ...) not read
*)
